// TIA Portal V18 export
TYPE "UDT_MEStoPLC_ext"
// stored: IsFailsafeCompliant false
   STRUCT
      Cmd : Struct
         "MES.Load_PartOK" : Bool;   // 查询事件反馈_OK/Loading part process - Part OK to assy all components
         "MES.Load_PartNG" : Bool;   // 查询事件反馈_NG/Loading part process - Part NOK to assy,check error code,fault and stop
         "MES.Load_2" : Bool;   // Loading part process - Spare
         "MES.Load_3" : Bool;   // Loading part process - Spare
         "MES.Unload_DataSaveOK" : Bool;   // 过程数据保存事件反馈_OK/Unloading part process - Results stored OK
         "MES.Unload_DataSaveNOK" : Bool;   // 过程数据保存事件反馈_NG/Unloading part process - Results stored NOK,check error code
         "MES.Unload_2" : Bool;   // Unloading part process - Spare
         "MES.Unload_3" : Bool;   // Unloading part process - Spare
         "MES.Spare8" : Bool;   // Spare - Future applications
         "MES.Spare9" : Bool;   // Spare - Future applications
         "MES.Spare10" : Bool;   // Spare - Future applications
         "MES.Spare11" : Bool;   // Spare - Future applications
         "MES.Spare12" : Bool;   // Spare - Future applications
         "MES.Spare13" : Bool;   // Spare - Future applications
         "MES.Spare14" : Bool;   // Spare - Future applications
         "MES.HeartbeatSignal" : Bool;   // MES心跳/MES TO PLC Heartbeat signal
      END_STRUCT;
   END_STRUCT;
END_TYPE
